FUNCTION_BLOCK FB_BHKW_Ablaufsteuerung
VAR_IN_OUT
	Zustand			: ST_BHKW_Zustand;
	Stellwert			: ST_BHKW_Stellwert;
END_VAR
VAR_INPUT
	Steuerung		: ST_BHKW_Steuerung;
	Parameter		: ST_BHKW_Parameter;
END_VAR
VAR_OUTPUT
END_VAR
VAR
	Timer			: TON;
END_VAR

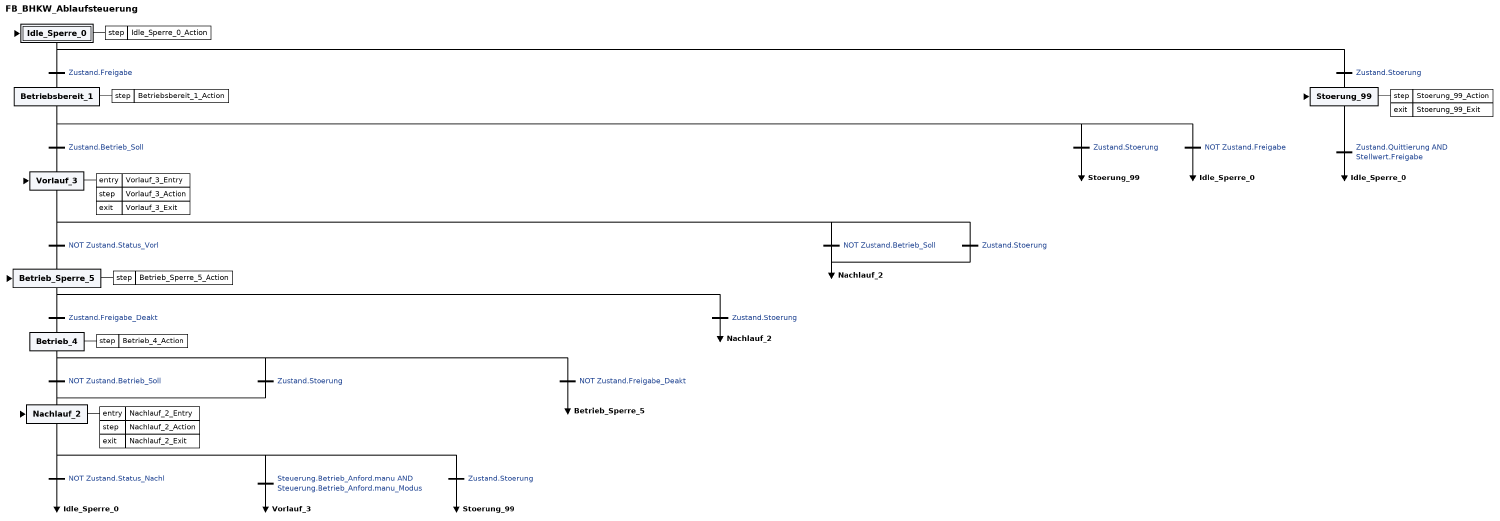
INITIAL_STEP Idle_Sperre_0:
    Idle_Sperre_0_Action(N);  // step action
END_STEP
TRANSITION FROM Idle_Sperre_0 TO Betriebsbereit_1
    := Zustand.Freigabe;
END_TRANSITION
TRANSITION FROM Idle_Sperre_0 TO Stoerung_99
    := Zustand.Stoerung;
END_TRANSITION
STEP Stoerung_99:
    Stoerung_99_Action(N);  // step action
    Stoerung_99_Exit(P0);  // exit action
END_STEP
TRANSITION FROM Stoerung_99 TO Idle_Sperre_0
    := Zustand.Quittierung AND Stellwert.Freigabe;
END_TRANSITION
STEP Betriebsbereit_1:
    Betriebsbereit_1_Action(N);  // step action
END_STEP
TRANSITION FROM Betriebsbereit_1 TO Vorlauf_3
    := Zustand.Betrieb_Soll;
END_TRANSITION
TRANSITION FROM Betriebsbereit_1 TO Stoerung_99
    := Zustand.Stoerung;
END_TRANSITION
TRANSITION FROM Betriebsbereit_1 TO Idle_Sperre_0
    := NOT Zustand.Freigabe;
END_TRANSITION
STEP Vorlauf_3:
    Vorlauf_3_Entry(P1);  // entry action
    Vorlauf_3_Action(N);  // step action
    Vorlauf_3_Exit(P0);  // exit action
END_STEP
TRANSITION FROM Vorlauf_3 TO Betrieb_Sperre_5
    := NOT Zustand.Status_Vorl;
END_TRANSITION
TRANSITION FROM Vorlauf_3 TO Nachlauf_2
    := NOT Zustand.Betrieb_Soll;
END_TRANSITION
TRANSITION FROM Vorlauf_3 TO Nachlauf_2
    := Zustand.Stoerung;
END_TRANSITION
STEP Betrieb_Sperre_5:
    Betrieb_Sperre_5_Action(N);  // step action
END_STEP
TRANSITION FROM Betrieb_Sperre_5 TO Betrieb_4
    := Zustand.Freigabe_Deakt;
END_TRANSITION
TRANSITION FROM Betrieb_Sperre_5 TO Nachlauf_2
    := Zustand.Stoerung;
END_TRANSITION
STEP Betrieb_4:
    Betrieb_4_Action(N);  // step action
END_STEP
TRANSITION FROM Betrieb_4 TO Nachlauf_2
    := NOT Zustand.Betrieb_Soll;
END_TRANSITION
TRANSITION FROM Betrieb_4 TO Nachlauf_2
    := Zustand.Stoerung;
END_TRANSITION
TRANSITION FROM Betrieb_4 TO Betrieb_Sperre_5
    := NOT Zustand.Freigabe_Deakt;
END_TRANSITION
STEP Nachlauf_2:
    Nachlauf_2_Entry(P1);  // entry action
    Nachlauf_2_Action(N);  // step action
    Nachlauf_2_Exit(P0);  // exit action
END_STEP
TRANSITION FROM Nachlauf_2 TO Idle_Sperre_0
    := NOT Zustand.Status_Nachl;
END_TRANSITION
TRANSITION FROM Nachlauf_2 TO Vorlauf_3
    := Steuerung.Betrieb_Anford.manu AND Steuerung.Betrieb_Anford.manu_Modus;
END_TRANSITION
TRANSITION FROM Nachlauf_2 TO Stoerung_99
    := Zustand.Stoerung;
END_TRANSITION

ACTION Betrieb_4_Action:
(* Stellwert setzen *)
Stellwert.Betrieb := TRUE;

(* Zustand setzen *)
Zustand.Status := E_BHKW_Zustand_Status_Betrieb;
END_ACTION

ACTION Betrieb_Sperre_5_Action:
(* Stellwert setzen *)
Stellwert.Betrieb := TRUE;

(* Zustand setzen *)
Zustand.Status := E_BHKW_Zustand_Status_Betrieb_Sperre;
END_ACTION

ACTION Betriebsbereit_1_Action:
(* Stellwert setzen *)
Stellwert.Betrieb := FALSE;
Stellwert.Freigabe := TRUE;

(* Zustand setzen *)
Zustand.Status := E_BHKW_Zustand_Status_Betriebsbereit;
END_ACTION

ACTION Idle_Sperre_0_Action:
(* Stellwert setzen *)
Stellwert.Betrieb := FALSE;

(* Zustand setzen *)
Zustand.Status := E_BHKW_Zustand_Status_Idle_Sperre;
END_ACTION

ACTION Nachlauf_2_Action:
(* Nachlauf Timer starten *)
Timer( 	IN := Zustand.Status_Nachl,
		PT := DINT_TO_TIME(Parameter.Zeit_Nachl)
);
Zustand.Status_Nachl	:= NOT(Timer.Q AND NOT Zustand.Betrieb);

(* Stellwert setzen *)
Stellwert.Betrieb := FALSE;
Stellwert.Freigabe := FALSE;

(* Zustand setzen *)
Zustand.Status := E_BHKW_Zustand_Status_Nachl;
END_ACTION

ACTION Nachlauf_2_Entry:
Zustand.Status_Nachl := TRUE;
(* Reset Timer *)
Timer(IN := FALSE);
END_ACTION

ACTION Nachlauf_2_Exit:
Zustand.Status_Nachl := FALSE;
END_ACTION

ACTION Stoerung_99_Action:
(* Stellwert setzen *)
Stellwert.Betrieb := FALSE;

(* Zustand setzen *)
Zustand.Stoerung := TRUE;
Zustand.Status := E_BHKW_Zustand_Status_Stoerung;
END_ACTION

ACTION Stoerung_99_Exit:
Zustand.Stoerung	:= FALSE;
END_ACTION

ACTION Vorlauf_3_Action:
(* Vorlaufzeit Timer starten *)
Timer( 	IN := Zustand.Status_Vorl,
		PT := DINT_TO_TIME(Parameter.Zeit_Vorl)
);

(* Stellwert setzen *)
Stellwert.Betrieb := Timer.Q;
Zustand.Status_Vorl := NOT (Timer.Q AND Zustand.Betrieb);

(* Zustand setzen *)
Zustand.Status := E_BHKW_Zustand_Status_Vorl;
END_ACTION

ACTION Vorlauf_3_Entry:
Zustand.Status_Vorl := TRUE;
(* Reset Timer *)
Timer(IN := FALSE);
END_ACTION

ACTION Vorlauf_3_Exit:
Zustand.Status_Vorl := FALSE;
END_ACTION

END_FUNCTION_BLOCK

(* stored: Version 1.1.0.1, ProductVersion 3.1.4024.9
   POU FB_BHKW_Ablaufsteuerung: Id {5ca6919c-a386-4a6e-a22c-395cdc7606ef}, SpecialFunc None
   Action Betrieb_4_Action: Id {c14b8b8f-a54a-4d03-a0b6-bebc780a5833}
   Action Betrieb_Sperre_5_Action: Id {e47498b7-d3f6-46d0-b013-022933ff753b}
   Action Betriebsbereit_1_Action: Id {40d03f8d-7eb2-4a5a-8253-799d50bfbeee}
   Action Idle_Sperre_0_Action: Id {05525993-c18b-4a8c-b33b-df9a340af7f9}
   Action Nachlauf_2_Action: Id {b14ae636-ce42-49b2-8775-3be10267f4dd}
   Action Nachlauf_2_Entry: Id {8de0ed36-0e65-4750-95b6-9e185f80ed76}
   Action Nachlauf_2_Exit: Id {1c1ea650-cf9d-45a6-850a-330ff9b1795f}
   Action Stoerung_99_Action: Id {ce45ab7a-2cb6-4c64-becd-81b2bda343b3}
   Action Stoerung_99_Exit: Id {29a5cab0-5613-4557-8b37-d5ce8bb4d3b0}
   Action Vorlauf_3_Action: Id {a15acd8d-7509-4095-bb56-fefba0e630fe}
   Action Vorlauf_3_Entry: Id {5bdcf7a9-f979-4eb9-88d2-e0b0f54e8f9f}
   Action Vorlauf_3_Exit: Id {2e725faf-a0c0-4b22-a3ba-342c59ddff98} *)
